{region '#Template'}
	{attribute 'Version' := '1.0.0.0'}
	{attribute 'Tags' := '"LCID": "1031", "Text": "GVL, DPAD, Trades, ObjectName, Description"'}
	{attribute 'Tags' := '"LCID": "1033", "Text": "GVL, DPAD, Trades, ObjectName, Description"'}
	{attribute 'Description' := '"LCID": "1031", "Text": "Textliste Gewerke"'}
	{attribute 'Description' := '"LCID": "1033", "Text": "Text list trades"'}
{endregion}

{attribute 'global_init_slot' := '40510'}
VAR_GLOBAL
  TxtTrade_Doors_gates_windows_sun_protection_sObjectName                :T_BA_StateText:='Doors, gates, windows, sun protection';
  TxtTrade_Doors_gates_windows_sun_protection_sDescription                :T_BA_StateText:='DGW';
  TxtTrade_Sewage_water_and_gas_plants_sObjectName                       :T_BA_StateText:='Sewage, water and gas plants';
  TxtTrade_Sewage_water_and_gas_plants_sDescription                       :T_BA_StateText:='SWG';
  TxtTrade_Heat_supply_systems_sObjectName                               :T_BA_StateText:='Heat supply systems';
  TxtTrade_Heat_supply_systems_sDescription                               :T_BA_StateText:='HTG';
  TxtTrade_Air_conditioning_sObjectName                                  :T_BA_StateText:='Air conditioning';
  TxtTrade_Air_conditioning_sDescription                                  :T_BA_StateText:='AC_';
  TxtTrade_Refrigeration_systems_sObjectName                             :T_BA_StateText:='Refrigeration systems';
  TxtTrade_Refrigeration_systems_sDescription                             :T_BA_StateText:='RFG';
  TxtTrade_High_voltage_systems_sObjectName                              :T_BA_StateText:='High-voltage systems';
  TxtTrade_High_voltage_systems_sDescription                              :T_BA_StateText:='HVS';
  TxtTrade_Telecommunication_and_information_technology_sObjectName      :T_BA_StateText:='Telecom. and information tech. equipment';
  TxtTrade_Telecommunication_and_information_technology_sDescription      :T_BA_StateText:='TIT';
  TxtTrade_Hazard_detection_and_alarm_systems_sObjectName                :T_BA_StateText:='Hazard detection and alarm systems';
  TxtTrade_Hazard_detection_and_alarm_systems_sDescription                :T_BA_StateText:='HDA';
  TxtTrade_Conveyors_sObjectName                                         :T_BA_StateText:='Conveyors';
  TxtTrade_Conveyors_sDescription                                         :T_BA_StateText:='CVY';
  TxtTrade_Kitchen_technology_systems_sObjectName                        :T_BA_StateText:='Kitchen technology systems';
  TxtTrade_Kitchen_technology_systems_sDescription                        :T_BA_StateText:='KTS';
  TxtTrade_Laundry_and_cleaning_systems_sObjectName                      :T_BA_StateText:='Laundry and cleaning systems';
  TxtTrade_Laundry_and_cleaning_systems_sDescription                      :T_BA_StateText:='LCS';
  TxtTrade_Media_supply_systems_sObjectName                              :T_BA_StateText:='Media supply systems';
  TxtTrade_Media_supply_systems_sDescription                              :T_BA_StateText:='MSS';
  TxtTrade_Medical_and_laboratory_equipment_sObjectName                  :T_BA_StateText:='Medical and laboratory equipment';
  TxtTrade_Medical_and_laboratory_equipment_sDescription                  :T_BA_StateText:='MED';
  TxtTrade_Fire_extinguishing_systems_sObjectName                        :T_BA_StateText:='Fire extinguishing systems';
  TxtTrade_Fire_extinguishing_systems_sDescription                        :T_BA_StateText:='FES';
  TxtTrade_Bathing_facilities_sObjectName                                :T_BA_StateText:='Bathing facilities';
  TxtTrade_Bathing_facilities_sDescription                                :T_BA_StateText:='BTF';
  TxtTrade_Process_heating_cooling_and_air_systems_sObjectName           :T_BA_StateText:='Process heating, cooling and air systems';
  TxtTrade_Process_heating_cooling_and_air_systems_sDescription           :T_BA_StateText:='PRO';
  TxtTrade_Waste_disposal_facilities_sObjectName                         :T_BA_StateText:='Waste disposal facilities';
  TxtTrade_Waste_disposal_facilities_sDescription                         :T_BA_StateText:='WDF';
  TxtTrade_Building_automation_and_control_systems_general_sObjectName   :T_BA_StateText:='Building automation  general';
  TxtTrade_Building_automation_and_control_systems_general_sDescription   :T_BA_StateText:='BAG';
  TxtTrade_Automation_focal_point_information_focal_point_sObjectName    :T_BA_StateText:='Automation focal point';
  TxtTrade_Automation_focal_point_information_focal_point_sDescription    :T_BA_StateText:='AFP';
  TxtTrade_Room_automation_sObjectName                                   :T_BA_StateText:='Room automation';
  TxtTrade_Room_automation_sDescription                                   :T_BA_StateText:='ROM';
  TxtTrade_Outdoor_devices_sObjectName                                   :T_BA_StateText:='Outdoor devices';
  TxtTrade_Outdoor_devices_sDescription                                   :T_BA_StateText:='ODD';
END_VAR

(* stored: Version 1.1.0.1, ProductVersion 3.1.4024.9
   GVL TxtTrade_1033: Id {d119fb7a-f21c-42a9-9365-2962eed09da3} *)
